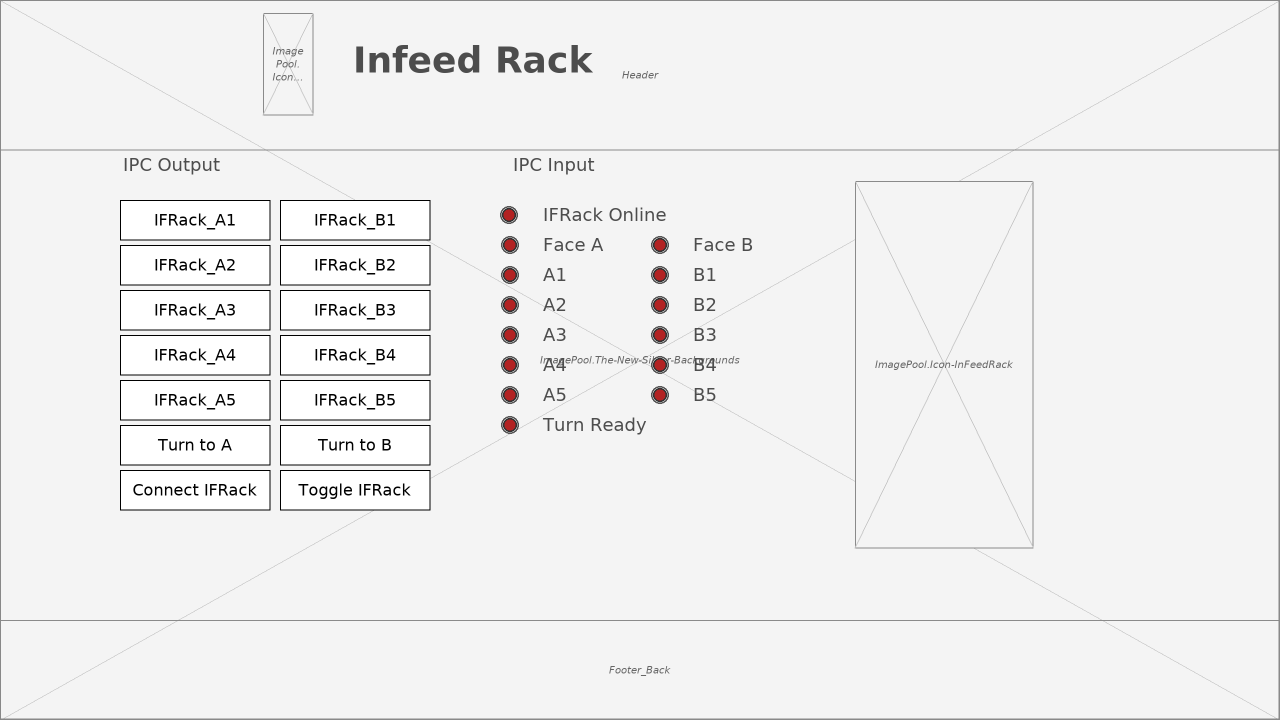
VISUALIZATION PAGE_InfeedRack  // 1280x720
    Image (0,0 1280x720), image: ImagePool.The-New-Silver-Backgrounds
    Frame (0,620 1280x100)
        shows Footer_Back()
    Frame (0,0 1280x150)
        shows Header()
    Label (350,40 300x40), "Infeed Rack"
    Label (120,150 150x30), "IPC Output"
    RoundedRectangle (120,200 150x40), "IFRack_A1"
        toggle INFEED_RACK.A1_Valve
    RoundedRectangle (120,245 150x40), "IFRack_A2"
        toggle INFEED_RACK.A2_Valve
    RoundedRectangle (120,290 150x40), "IFRack_A3"
        toggle INFEED_RACK.A3_Valve
    RoundedRectangle (120,335 150x40), "IFRack_A4"
        toggle INFEED_RACK.A4_Valve
    RoundedRectangle (120,380 150x40), "IFRack_A5"
        toggle INFEED_RACK.A5_Valve
    RoundedRectangle (280,200 150x40), "IFRack_B1"
        toggle INFEED_RACK.B1_Valve
    RoundedRectangle (280,245 150x40), "IFRack_B2"
        toggle INFEED_RACK.B2_Valve
    RoundedRectangle (280,290 150x40), "IFRack_B3"
        toggle INFEED_RACK.B3_Valve
    RoundedRectangle (280,335 150x40), "IFRack_B4"
        toggle INFEED_RACK.B4_Valve
    RoundedRectangle (280,380 150x40), "IFRack_B5"
        toggle INFEED_RACK.B5_Valve
    RoundedRectangle (120,425 150x40), "Turn to A"
        toggle INFEED_RACK.Turn_B_to_A
    RoundedRectangle (280,425 150x40), "Turn to B"
        toggle INFEED_RACK.Turn_A_to_B
    RoundedRectangle (120,470 150x40), "Connect IFRack"
        toggle INFEED_RACK.IFRack_Connect
    RoundedRectangle (280,470 150x40), "Toggle IFRack"
        tap INFEED_RACK.bstart_Write
    Label (510,150 150x30), "IPC Input"
    Label (540,380 100x30), "A5"
    Label (690,380 100x30), "B5"
    Label (540,200 130x30), "IFRack Online"
    Lamp1 (499,205 20x20), variable: INFEED_RACK.IFRack_Ready, style: Lamp-Lamp1-Red
    Lamp1 (500,235 20x20), variable: INFEED_RACK.FaceA_InWC, style: Lamp-Lamp1-Red
    Lamp1 (500,265 20x20), variable: INFEED_RACK.A1_Sensor, style: Lamp-Lamp1-Red
    Lamp1 (500,295 20x20), variable: INFEED_RACK.A2_Sensor, style: Lamp-Lamp1-Red
    Lamp1 (500,325 20x20), variable: INFEED_RACK.A3_Sensor, style: Lamp-Lamp1-Red
    Label (540,260 100x30), "A1"
    Label (540,290 100x30), "A2"
    Label (540,320 100x30), "A3"
    Label (540,350 100x30), "A4"
    Lamp1 (500,355 20x20), variable: INFEED_RACK.A4_Sensor, style: Lamp-Lamp1-Red
    Lamp1 (500,385 20x20), variable: INFEED_RACK.A5_Sensor, style: Lamp-Lamp1-Red
    Label (540,230 100x30), "Face A"
    Lamp1 (650,235 20x20), variable: INFEED_RACK.FaceB_InWC, style: Lamp-Lamp1-Red
    Lamp1 (650,265 20x20), variable: INFEED_RACK.B1_Sensor, style: Lamp-Lamp1-Red
    Lamp1 (650,295 20x20), variable: INFEED_RACK.B2_Sensor, style: Lamp-Lamp1-Red
    Lamp1 (650,325 20x20), variable: INFEED_RACK.B3_Sensor, style: Lamp-Lamp1-Red
    Label (690,260 100x30), "B1"
    Label (690,290 100x30), "B2"
    Label (690,320 100x30), "B3"
    Label (690,350 100x30), "B4"
    Lamp1 (650,355 20x20), variable: INFEED_RACK.B4_Sensor, style: Lamp-Lamp1-Red
    Lamp1 (650,385 20x20), variable: INFEED_RACK.B5_Sensor, style: Lamp-Lamp1-Red
    Label (690,230 100x30), "Face B"
    Image (263,13 50x102), image: ImagePool.Icon-InFeedRack
    Image (855,181 178x367), image: ImagePool.Icon-InFeedRack
    Lamp1 (500,415 20x20), variable: INFEED_RACK.IFRack_TurnReady, style: Lamp-Lamp1-Red
    Label (540,410 127x30), "Turn Ready"
END_VISUALIZATION

(* stored: Version 1.1.0.1, ProductVersion 3.1.4024.12
   Visu PAGE_InfeedRack: Id {f983bf0a-d8a0-4718-b72f-fb237930ea94} *)
